Fanuc KAREL source: kx00002.KL

-- PROVISIONAL review KL for V1013-1; original PC SHA256 b25ecb5062d861ed8447f028f19d9bc94bcb28f012d881d32fda251ae2710227
-- Incomplete behavior may be omitted. Consult companion uncertainty JSON. Do not deploy.
PROGRAM KX00002
%NOLOCKGROUP
VAR
  I : INTEGER
  J : INTEGER
  B : BOOLEAN
  F : FILE
  S : STRING[80]
-- UNRESOLVED_DECL P type=000102
BEGIN
  -- UNRESOLVED_PC offsets 5-32; opcodes 22,3F,3F,3D
  -- UNRESOLVED_PC offsets 37-44; opcodes 22,39
  -- UNRESOLVED_PC offsets 49-53; opcodes 7F
END KX00002
